(* CODESYS project OOP example Polymorphism.project

Project tree, tasks and I/O mapping:
  Device : CODESYS Control for Raspberry Pi SL, 3S - Smart Software Solutions GmbH, version 3.5.12.30
    application Application
      libraries: Standard, * (System); VisuDialogs, * (System); SysFile, 3.5.9.0 (System); AlarmManager, 3.5.12.0 (Intern)
      task MainTask (cyclic, interval 500 ms, priority 1, watchdog 1000 ms x 1) calls Polymorphism
      program Polymorphism [ST]
    SoftMotion General Axis Pool
    I²C
    SPI
    GPIOs_A_B : GPIOs B+/Pi2, 3S - Smart Software Solutions GmbH, version 3.5.11.0
        unmapped channels: digital inputs (GPIO0..GPIO31), digital outputs (GPIO0..GPIO31)
    Onewire
    Camera device
      <Empty>
  libraries: VisuSymbols, 3.5.10.0 (System)
  Polymorphism/
    function block FB_Engine [ST]: Start, Stop, MaxVelocity, Temperature, Velocity
    function block FB_NewEngine [ST]: Gear, Start
*)

// Device/Application/Polymorphism
PROGRAM Polymorphism
VAR
	fbEngine : FB_Engine;
	fbNewEngine : FB_NewEngine;
	
	xSwitchEngine : BOOL;
	refEngine : REFERENCE TO FB_Engine := fbEngine; // reference to baseclass
	
	rTemperature : REAL;
	xStart : BOOL := TRUE;
	rMaxVelocity : REAL := 130; //kmph
	rVelocity : REAL := 100; //kmph
	iGear : INT  := 5;
	xIsStarted : BOOL;
	xStopped : BOOL;
END_VAR

// polymorphism  (greek for 'has many forms') = ambiguity 
// The reference refEngine can take any FB that is derived from the baseclass, so in this example FB_Engine and FB_NewEngine
IF NOT xSwitchEngine THEN
   refEngine REF= fbEngine;
ELSE
   refEngine REF= fbNewEngine;
END_IF
  
IF xStart THEN
    xIsStarted := refEngine.Start(rVelocity,iGear);
	xStopped := FALSE;
ELSE 
	xIsStarted := FALSE;
    xStopped := refEngine.Stop(); 
END_IF

refEngine.MaxVelocity := rMaxVelocity;
rTemperature := refEngine.Temperature;  

xStart := NOT xStart;

END_PROGRAM

// Polymorphism/FB_Engine
// Class FB_Engine
FUNCTION_BLOCK FB_Engine
VAR
   _xStarted : BOOL;
   _rVelocity : REAL;
   _rMaxVelocity : REAL;
   _iGear : INT;
   _rTemperature : REAL;
END_VAR

//The THIS pointer is available to all function blocks and points to the current function block instance. 
//It is required whenever a method contains a local variable which obscures a variable in the function block.
//
//An assignment statement within the method sets the value of the local variable. 
//If we want the method to set the value of the local variable in the function block, we need to use the THIS pointer to access it.
METHOD Start : Bool;
VAR_INPUT
   rVelocity : REAL;
   iGear     : INT;
END_VAR
THIS^._xStarted  := TRUE;
Start            := TRUE;
THIS^._iGear     := iGear;
THIS^._rVelocity := MIN( ABS(THIS^._rMaxVelocity), rVelocity );

CASE TO_INT( THIS^._rVelocity ) OF // implicit typecasting(TO_INT), use REAL_TO_INT for explicit typecasting
   0..100 :
      THIS^._rTemperature := 50;
   101..1000:
      THIS^._rTemperature := 90;
   1001..10000:
      THIS^._rTemperature := 100;
   10001..32767:
      THIS^._rTemperature := 150;
END_CASE
END_METHOD

METHOD Stop : BOOL
VAR_INPUT
END_VAR
THIS^._xStarted := FALSE;
Stop            := TRUE;
END_METHOD

PROPERTY MaxVelocity : REAL
SET
THIS^._rMaxVelocity := MaxVelocity;
END_SET
GET
MaxVelocity := THIS^._rMaxVelocity;
END_GET
END_PROPERTY

PROPERTY Temperature : REAL
GET
Temperature := THIS^._rTemperature;
END_GET
END_PROPERTY

PROPERTY Velocity : real
GET
Velocity := THIS^._rVelocity;
END_GET
END_PROPERTY

END_FUNCTION_BLOCK

// Polymorphism/FB_NewEngine
FUNCTION_BLOCK FB_NewEngine EXTENDS FB_Engine

// HAS GOT 2 NEW Features;
// 1) START has been redefined and 
// 2) A new Gear accessor has been added
//
// these methods are fixed to the class
SUPER^();

// new property to get / set the gear after start
PROPERTY Gear : int
SET
THIS^._iGear := Gear;
END_SET
GET
Gear := THIS^._iGear;
END_GET
END_PROPERTY

METHOD Start : BOOL;
VAR_INPUT
   fVelocity : REAL;
   nGear     : INT;
END_VAR
// Overwriting an existing method (OVERRIDE)

// new: setting gear via property Gear setter
SUPER^.Start(nGear, TO_INT(fVelocity)); // calls Start() of FB_Engine, see below for explanation
Gear := nGear;


// SUPER^. POINTER
//In the above example, we created a new Start() METHOD in FB_NewEngine 
//and copied the existing code from FB_Engine into the new method. 
//This is not always possible, and it also runs counter to the principle of reuse!
//
//Consequently, every function block which is derived from another function block has access to a pointer called SUPER. 
//This can be used to access elements (methods, properties, local variables, etc.) from the parent function block.
//
//
//SUPER^.Start(nGear, fVelocity); // calls Start() of FB_Engine
//Gear := nGear;
//
//Instead of copying code from the parent function block to the new method, 
//the SUPER pointer can be used to call the method from the FB_Engine function block. 
//This does away with the need to copy the code. 
//So, SUPER calls the Father of a method
END_METHOD

END_FUNCTION_BLOCK
